TYPE T_DefectErrorID : STRING(4); END_TYPE

(* stored: Version 1.1.0.1, ProductVersion 3.1.4024.12
   DUT T_DefectErrorID: Id {25d2ecbb-beff-4a96-8332-2c603fbfc68b} *)
